FUNCTION_BLOCK TestCSVLogger EXTENDS TcUnit.FB_TestSuite
VAR_INPUT
END_VAR
VAR_OUTPUT
END_VAR
VAR
END_VAR

submit_alarm();

METHOD submit_alarm
VAR_INPUT
END_VAR
VAR_INST
  sut: CSVLoggerTestsystem;
  state_number: INT;
END_VAR
TEST('Submit alarm');

sut.logging.run();

CASE state_number OF
0:
  IF sut.logging.time_valid THEN
    state_number := state_number + 10;
	END_IF
10:
  sut.logger.path := 'C:\';
  sut.logging.add_logger(sut.logger);
  sut.event.message := 'Alarm';
  sut.event.alarm();
  state_number := state_number + 10;
20:
  IF sut.logger.state_number = 0 THEN
    TEST_FINISHED();
	END_IF
END_CASE
END_METHOD

END_FUNCTION_BLOCK

(* stored: Version 1.1.0.1, ProductVersion 3.1.4024.9
   POU TestCSVLogger: Id {6eb9b79c-7996-4180-884f-6c85712e4467}, SpecialFunc None
   Method submit_alarm: Id {d77c3969-9108-4692-b556-3c4076a29c72} *)
